TYPE ST_PLCstate_get :
STRUCT
	r_CPUload		: REAL;
	e_ProfinetState	: eNetcomState;
	e_EthercatState	: eNetcomState;
END_STRUCT
END_TYPE

(* stored: Version 1.1.0.1, ProductVersion 3.1.4024.12
   DUT ST_PLCstate_get: Id {385ab9d8-daee-44b8-8805-2cc838d355f3} *)
